// TIA Portal V20 export
TYPE "LKinCtrl_PathEditor_typeLinkTableExternalEvents"
// stored: Access Published
   STRUCT
      selectionChanged { ExternalAccessible := 'False'; ExternalVisible := 'False'; ExternalWritable := 'False'} : Struct
         trigger : Bool;   // triggers event. Reset internally.
         selectedIndex : DInt := -1;   // Selected index in table. Only valid if noSelection = FALSE.
         noSelection : Bool := true;   // TRUE: nothing is selected in table.
         contentType : Int;   // 10: variables, 11: conditions, 12: Inputs, 13: Outputs, 14: Points, 20: Axes, 21: PosSyncAxes , 22: SyncAxes, 30: Labels, 40: Sequences
      END_STRUCT;
      updatePathTable { ExternalAccessible := 'False'; ExternalVisible := 'False'; ExternalWritable := 'False'} : Bool;
   END_STRUCT;
END_TYPE
